// TIA Portal V19 export
FUNCTION "MODE SELECTION" : Void   // FC3, LAD
{ S7_Optimized_Access := 'TRUE' }
// stored: SetENOAutomatically false
   VAR_TEMP   // added for the SCL form of the ladder/FBD networks
      _w1 : Bool;
   END_VAR
BEGIN

REGION Network 1: STANDBY \///////////////////////////////// RO-1 ///////////////////////////////////////////
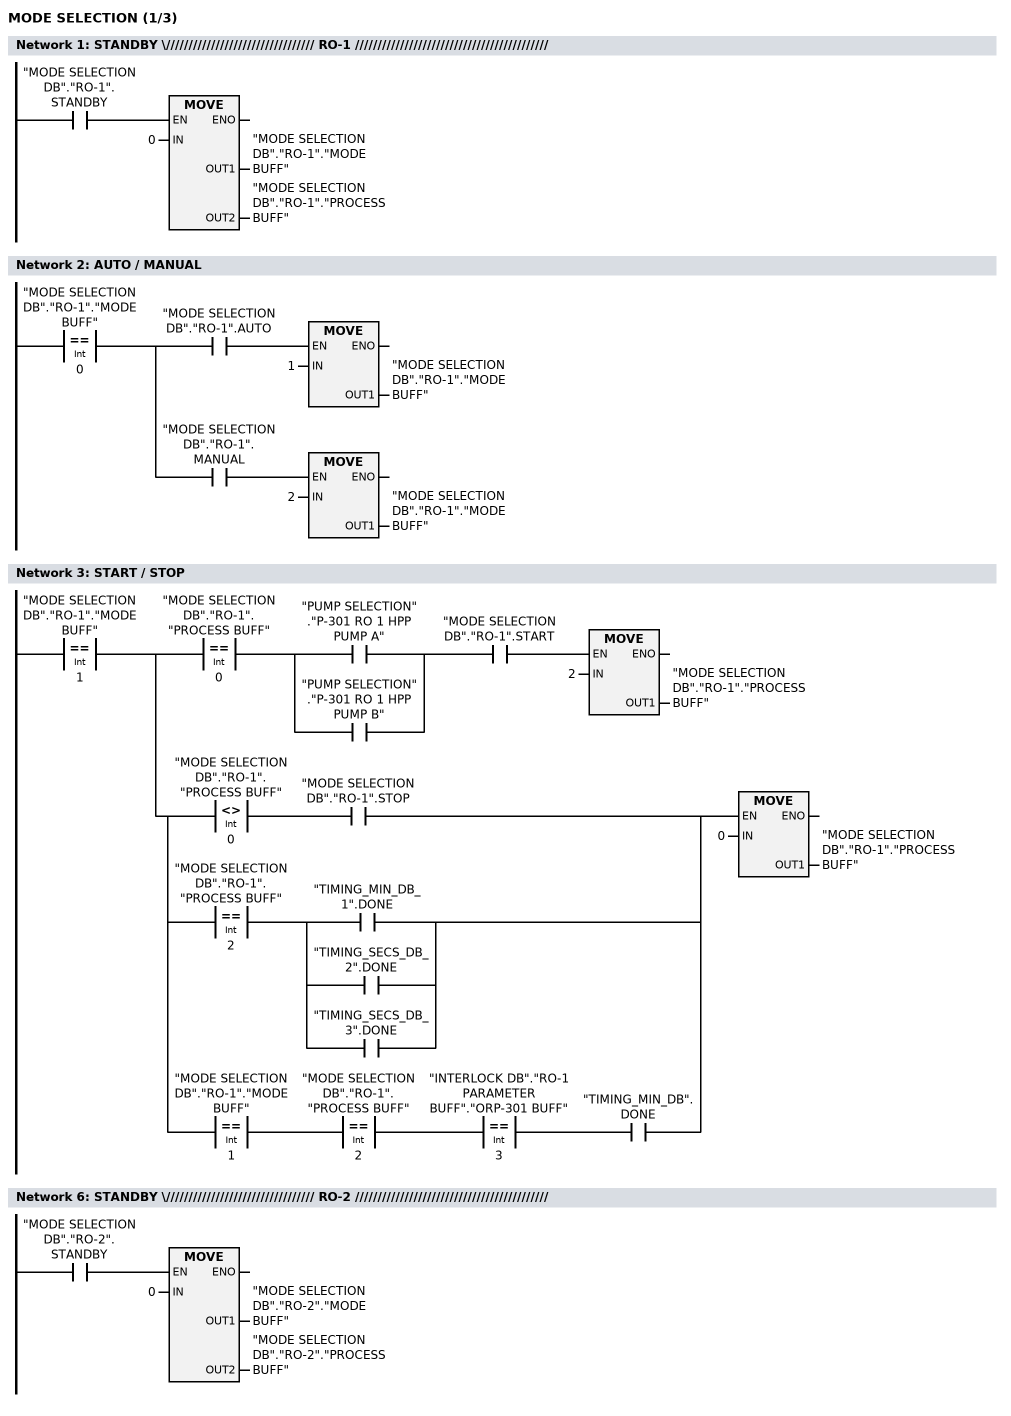
   RUNG wire#powerrail
      Contact( "MODE SELECTION DB"."RO-1".STANDBY )
      Move(in := 0, out1 => "MODE SELECTION DB"."RO-1"."MODE BUFF", out2 => "MODE SELECTION DB"."RO-1"."PROCESS BUFF")
   END_RUNG
   // the same network as SCL:
   IF "MODE SELECTION DB"."RO-1".STANDBY THEN
       "MODE SELECTION DB"."RO-1"."MODE BUFF" := 0;
       "MODE SELECTION DB"."RO-1"."PROCESS BUFF" := 0;
   END_IF;
END_REGION

REGION Network 2: AUTO / MANUAL
   RUNG wire#powerrail
      { S7_Templates := "SrcType := Int" } EQ_Contact(in1 := "MODE SELECTION DB"."RO-1"."MODE BUFF", in2 := 0)
      wire#w1
      Contact( "MODE SELECTION DB"."RO-1".AUTO )
      Move(in := 1, out1 => "MODE SELECTION DB"."RO-1"."MODE BUFF")
   END_RUNG
   RUNG wire#w1
      Contact( "MODE SELECTION DB"."RO-1".MANUAL )
      Move(in := 2, out1 => "MODE SELECTION DB"."RO-1"."MODE BUFF")
   END_RUNG
   // the same network as SCL:
   #_w1 := "MODE SELECTION DB"."RO-1"."MODE BUFF" = 0;
   IF #_w1 AND "MODE SELECTION DB"."RO-1".AUTO THEN "MODE SELECTION DB"."RO-1"."MODE BUFF" := 1; END_IF;
   IF #_w1 AND "MODE SELECTION DB"."RO-1".MANUAL THEN "MODE SELECTION DB"."RO-1"."MODE BUFF" := 2; END_IF;
END_REGION

REGION Network 3: START / STOP
   RUNG wire#powerrail
      { S7_Templates := "SrcType := Int" } EQ_Contact(in1 := "MODE SELECTION DB"."RO-1"."MODE BUFF", in2 := 1)
      wire#w1
      { S7_Templates := "SrcType := Int" } EQ_Contact(in1 := "MODE SELECTION DB"."RO-1"."PROCESS BUFF", in2 := 0)
      wire#w2
      Contact( "PUMP SELECTION"."P-301 RO 1 HPP PUMP A" )
      wire#w3
      Contact( "MODE SELECTION DB"."RO-1".START )
      Move(in := 2, out1 => "MODE SELECTION DB"."RO-1"."PROCESS BUFF")
   END_RUNG
   RUNG wire#w2
      Contact( "PUMP SELECTION"."P-301 RO 1 HPP PUMP B" )
   END_RUNG wire#w3
   RUNG wire#w1
      { S7_Templates := "SrcType := Int" } NE_Contact(in1 := "MODE SELECTION DB"."RO-1"."PROCESS BUFF", in2 := 0)
      Contact( "MODE SELECTION DB"."RO-1".STOP )
      wire#w4
      Move(in := 0, out1 => "MODE SELECTION DB"."RO-1"."PROCESS BUFF")
   END_RUNG
   RUNG wire#w1
      { S7_Templates := "SrcType := Int" } EQ_Contact(in1 := "MODE SELECTION DB"."RO-1"."PROCESS BUFF", in2 := 2)
      wire#w5
      Contact( "TIMING_MIN_DB_1".DONE )
   END_RUNG wire#w4
   RUNG wire#w5
      Contact( "TIMING_SECS_DB_2".DONE )
   END_RUNG wire#w4
   RUNG wire#w5
      Contact( "TIMING_SECS_DB_3".DONE )
   END_RUNG wire#w4
   RUNG wire#w1
      { S7_Templates := "SrcType := Int" } EQ_Contact(in1 := "MODE SELECTION DB"."RO-1"."MODE BUFF", in2 := 1)
      { S7_Templates := "SrcType := Int" } EQ_Contact(in1 := "MODE SELECTION DB"."RO-1"."PROCESS BUFF", in2 := 2)
      { S7_Templates := "SrcType := Int" } EQ_Contact(in1 := "INTERLOCK DB"."RO-1 PARAMETER BUFF"."ORP-301 BUFF", in2 := 3)
      Contact( "TIMING_MIN_DB".DONE )
   END_RUNG wire#w4
   // the same network as SCL:
   #_w1 := "MODE SELECTION DB"."RO-1"."MODE BUFF" = 1;
   IF #_w1 AND ("MODE SELECTION DB"."RO-1"."PROCESS BUFF" = 0) AND ("PUMP SELECTION"."P-301 RO 1 HPP PUMP A" OR "PUMP SELECTION"."P-301 RO 1 HPP PUMP B") AND "MODE SELECTION DB"."RO-1".START THEN
       "MODE SELECTION DB"."RO-1"."PROCESS BUFF" := 2;
   END_IF;
   IF #_w1 AND ((("MODE SELECTION DB"."RO-1"."PROCESS BUFF" <> 0) AND "MODE SELECTION DB"."RO-1".STOP) OR (("MODE SELECTION DB"."RO-1"."PROCESS BUFF" = 2) AND ("TIMING_MIN_DB_1".DONE OR "TIMING_SECS_DB_2".DONE OR "TIMING_SECS_DB_3".DONE)) OR (("MODE SELECTION DB"."RO-1"."MODE BUFF" = 1) AND ("MODE SELECTION DB"."RO-1"."PROCESS BUFF" = 2) AND ("INTERLOCK DB"."RO-1 PARAMETER BUFF"."ORP-301 BUFF" = 3) AND "TIMING_MIN_DB".DONE)) THEN
       "MODE SELECTION DB"."RO-1"."PROCESS BUFF" := 0;
   END_IF;
END_REGION

REGION Network 6: STANDBY \///////////////////////////////// RO-2 ///////////////////////////////////////////
   RUNG wire#powerrail
      Contact( "MODE SELECTION DB"."RO-2".STANDBY )
      Move(in := 0, out1 => "MODE SELECTION DB"."RO-2"."MODE BUFF", out2 => "MODE SELECTION DB"."RO-2"."PROCESS BUFF")
   END_RUNG
   // the same network as SCL:
   IF "MODE SELECTION DB"."RO-2".STANDBY THEN
       "MODE SELECTION DB"."RO-2"."MODE BUFF" := 0;
       "MODE SELECTION DB"."RO-2"."PROCESS BUFF" := 0;
   END_IF;
END_REGION

REGION Network 7: AUTO / MANUAL
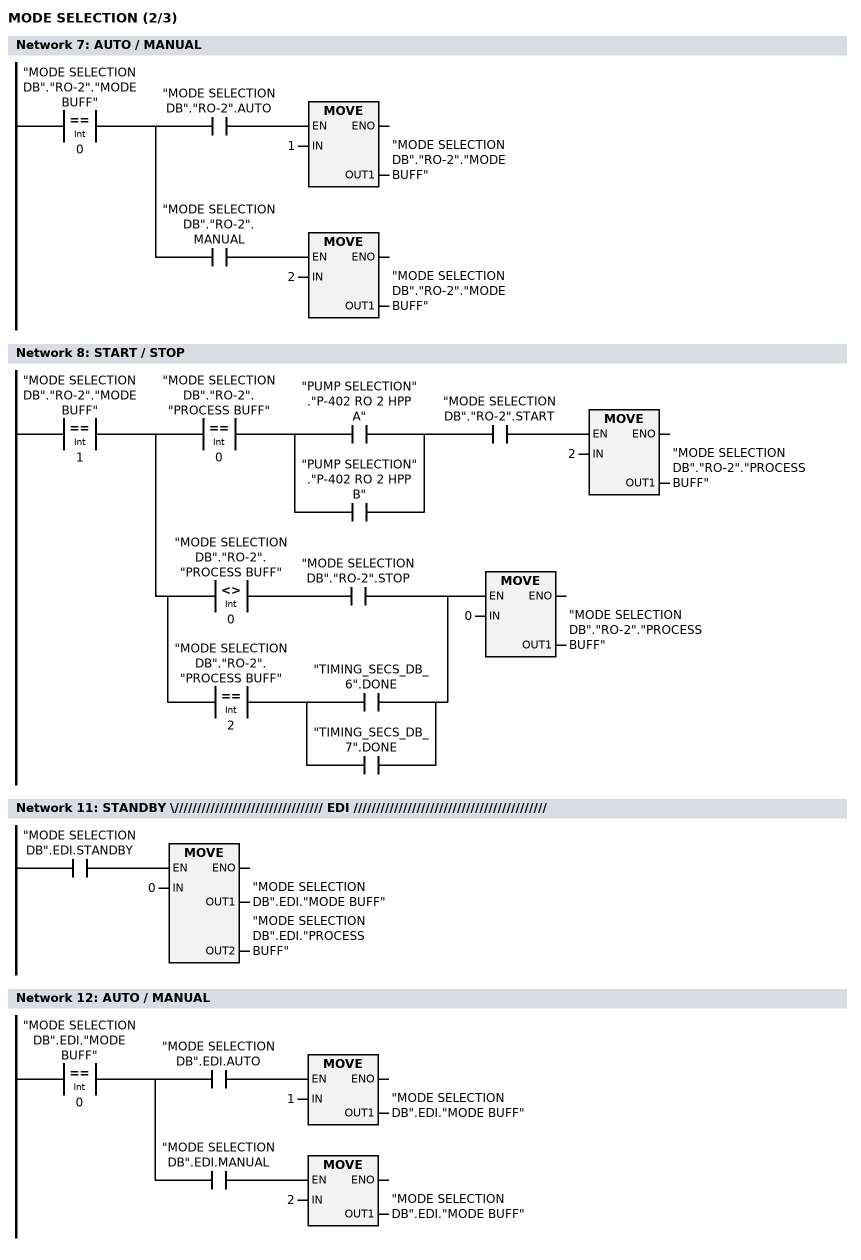
   RUNG wire#powerrail
      { S7_Templates := "SrcType := Int" } EQ_Contact(in1 := "MODE SELECTION DB"."RO-2"."MODE BUFF", in2 := 0)
      wire#w1
      Contact( "MODE SELECTION DB"."RO-2".AUTO )
      Move(in := 1, out1 => "MODE SELECTION DB"."RO-2"."MODE BUFF")
   END_RUNG
   RUNG wire#w1
      Contact( "MODE SELECTION DB"."RO-2".MANUAL )
      Move(in := 2, out1 => "MODE SELECTION DB"."RO-2"."MODE BUFF")
   END_RUNG
   // the same network as SCL:
   #_w1 := "MODE SELECTION DB"."RO-2"."MODE BUFF" = 0;
   IF #_w1 AND "MODE SELECTION DB"."RO-2".AUTO THEN "MODE SELECTION DB"."RO-2"."MODE BUFF" := 1; END_IF;
   IF #_w1 AND "MODE SELECTION DB"."RO-2".MANUAL THEN "MODE SELECTION DB"."RO-2"."MODE BUFF" := 2; END_IF;
END_REGION

REGION Network 8: START / STOP
   RUNG wire#powerrail
      { S7_Templates := "SrcType := Int" } EQ_Contact(in1 := "MODE SELECTION DB"."RO-2"."MODE BUFF", in2 := 1)
      wire#w1
      { S7_Templates := "SrcType := Int" } EQ_Contact(in1 := "MODE SELECTION DB"."RO-2"."PROCESS BUFF", in2 := 0)
      wire#w2
      Contact( "PUMP SELECTION"."P-402 RO 2 HPP A" )
      wire#w3
      Contact( "MODE SELECTION DB"."RO-2".START )
      Move(in := 2, out1 => "MODE SELECTION DB"."RO-2"."PROCESS BUFF")
   END_RUNG
   RUNG wire#w2
      Contact( "PUMP SELECTION"."P-402 RO 2 HPP B" )
   END_RUNG wire#w3
   RUNG wire#w1
      { S7_Templates := "SrcType := Int" } NE_Contact(in1 := "MODE SELECTION DB"."RO-2"."PROCESS BUFF", in2 := 0)
      Contact( "MODE SELECTION DB"."RO-2".STOP )
      wire#w4
      Move(in := 0, out1 => "MODE SELECTION DB"."RO-2"."PROCESS BUFF")
   END_RUNG
   RUNG wire#w1
      { S7_Templates := "SrcType := Int" } EQ_Contact(in1 := "MODE SELECTION DB"."RO-2"."PROCESS BUFF", in2 := 2)
      wire#w5
      Contact( "TIMING_SECS_DB_6".DONE )
   END_RUNG wire#w4
   RUNG wire#w5
      Contact( "TIMING_SECS_DB_7".DONE )
   END_RUNG wire#w4
   // the same network as SCL:
   #_w1 := "MODE SELECTION DB"."RO-2"."MODE BUFF" = 1;
   IF #_w1 AND ("MODE SELECTION DB"."RO-2"."PROCESS BUFF" = 0) AND ("PUMP SELECTION"."P-402 RO 2 HPP A" OR "PUMP SELECTION"."P-402 RO 2 HPP B") AND "MODE SELECTION DB"."RO-2".START THEN
       "MODE SELECTION DB"."RO-2"."PROCESS BUFF" := 2;
   END_IF;
   IF #_w1 AND ((("MODE SELECTION DB"."RO-2"."PROCESS BUFF" <> 0) AND "MODE SELECTION DB"."RO-2".STOP) OR (("MODE SELECTION DB"."RO-2"."PROCESS BUFF" = 2) AND ("TIMING_SECS_DB_6".DONE OR "TIMING_SECS_DB_7".DONE))) THEN
       "MODE SELECTION DB"."RO-2"."PROCESS BUFF" := 0;
   END_IF;
END_REGION

REGION Network 11: STANDBY \///////////////////////////////// EDI ///////////////////////////////////////////
   RUNG wire#powerrail
      Contact( "MODE SELECTION DB".EDI.STANDBY )
      Move(in := 0, out1 => "MODE SELECTION DB".EDI."MODE BUFF", out2 => "MODE SELECTION DB".EDI."PROCESS BUFF")
   END_RUNG
   // the same network as SCL:
   IF "MODE SELECTION DB".EDI.STANDBY THEN
       "MODE SELECTION DB".EDI."MODE BUFF" := 0;
       "MODE SELECTION DB".EDI."PROCESS BUFF" := 0;
   END_IF;
END_REGION

REGION Network 12: AUTO / MANUAL
   RUNG wire#powerrail
      { S7_Templates := "SrcType := Int" } EQ_Contact(in1 := "MODE SELECTION DB".EDI."MODE BUFF", in2 := 0)
      wire#w1
      Contact( "MODE SELECTION DB".EDI.AUTO )
      Move(in := 1, out1 => "MODE SELECTION DB".EDI."MODE BUFF")
   END_RUNG
   RUNG wire#w1
      Contact( "MODE SELECTION DB".EDI.MANUAL )
      Move(in := 2, out1 => "MODE SELECTION DB".EDI."MODE BUFF")
   END_RUNG
   // the same network as SCL:
   #_w1 := "MODE SELECTION DB".EDI."MODE BUFF" = 0;
   IF #_w1 AND "MODE SELECTION DB".EDI.AUTO THEN "MODE SELECTION DB".EDI."MODE BUFF" := 1; END_IF;
   IF #_w1 AND "MODE SELECTION DB".EDI.MANUAL THEN "MODE SELECTION DB".EDI."MODE BUFF" := 2; END_IF;
END_REGION

REGION Network 13: START / STOP
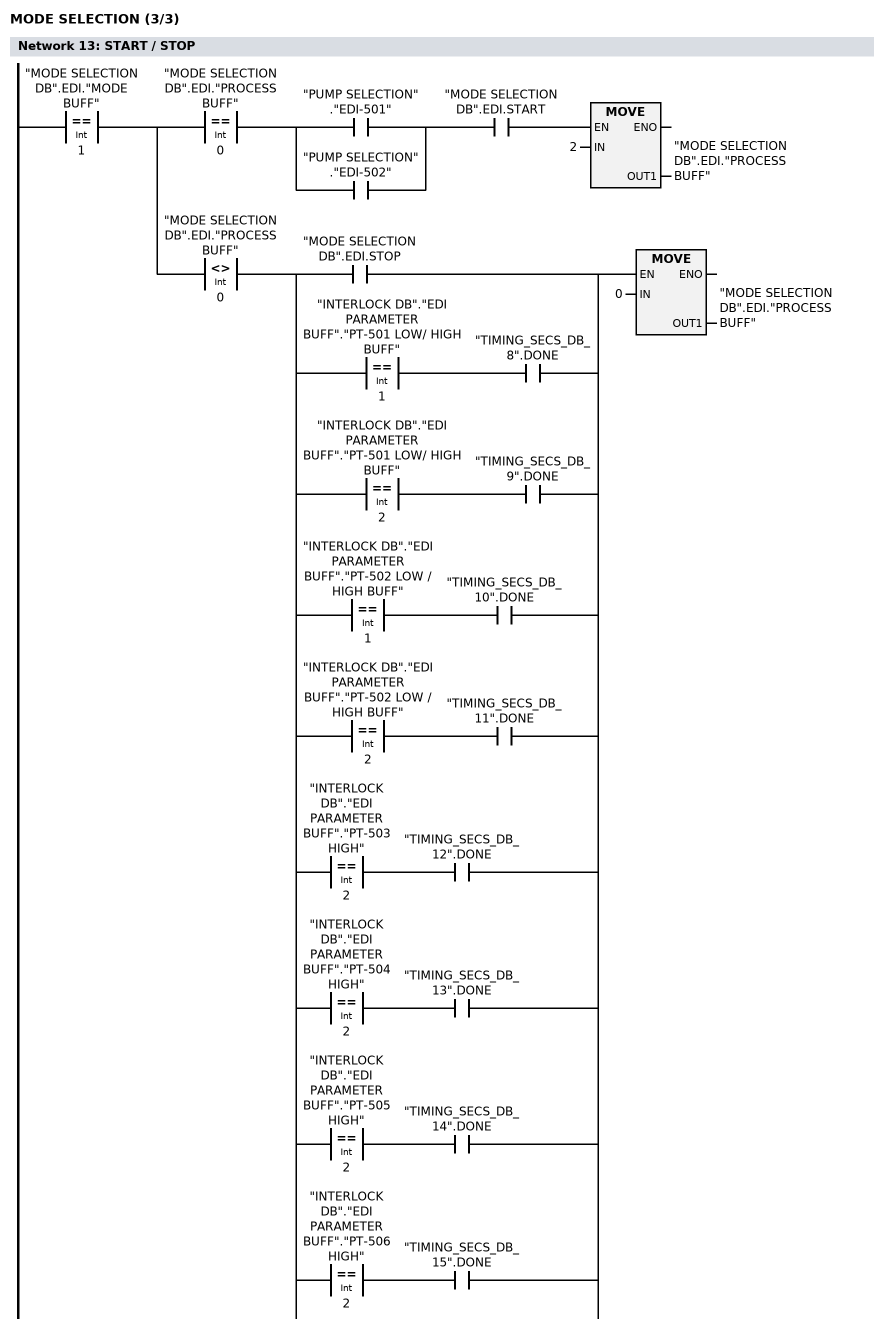
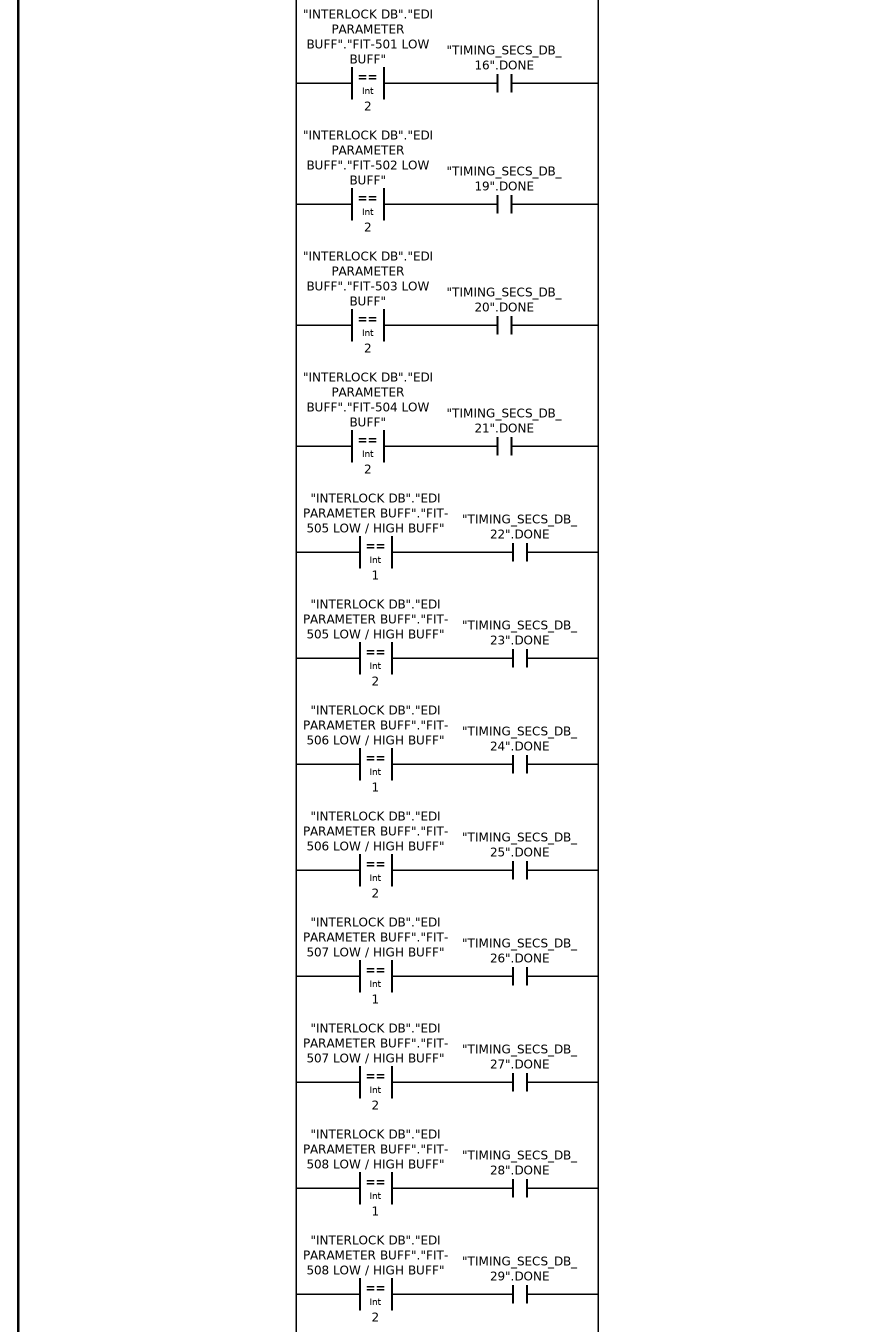
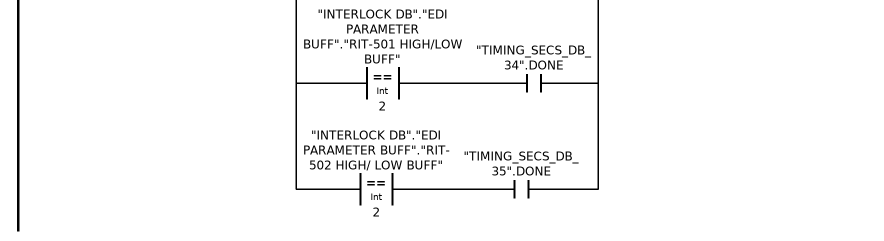
   RUNG wire#powerrail
      { S7_Templates := "SrcType := Int" } EQ_Contact(in1 := "MODE SELECTION DB".EDI."MODE BUFF", in2 := 1)
      wire#w1
      { S7_Templates := "SrcType := Int" } EQ_Contact(in1 := "MODE SELECTION DB".EDI."PROCESS BUFF", in2 := 0)
      wire#w2
      Contact( "PUMP SELECTION"."EDI-501" )
      wire#w3
      Contact( "MODE SELECTION DB".EDI.START )
      Move(in := 2, out1 => "MODE SELECTION DB".EDI."PROCESS BUFF")
   END_RUNG
   RUNG wire#w2
      Contact( "PUMP SELECTION"."EDI-502" )
   END_RUNG wire#w3
   RUNG wire#w1
      { S7_Templates := "SrcType := Int" } NE_Contact(in1 := "MODE SELECTION DB".EDI."PROCESS BUFF", in2 := 0)
      wire#w4
      Contact( "MODE SELECTION DB".EDI.STOP )
      wire#w5
      Move(in := 0, out1 => "MODE SELECTION DB".EDI."PROCESS BUFF")
   END_RUNG
   RUNG wire#w4
      { S7_Templates := "SrcType := Int" } EQ_Contact(in1 := "INTERLOCK DB"."EDI PARAMETER BUFF"."PT-501 LOW/ HIGH BUFF", in2 := 1)
      Contact( "TIMING_SECS_DB_8".DONE )
   END_RUNG wire#w5
   RUNG wire#w4
      { S7_Templates := "SrcType := Int" } EQ_Contact(in1 := "INTERLOCK DB"."EDI PARAMETER BUFF"."PT-501 LOW/ HIGH BUFF", in2 := 2)
      Contact( "TIMING_SECS_DB_9".DONE )
   END_RUNG wire#w5
   RUNG wire#w4
      { S7_Templates := "SrcType := Int" } EQ_Contact(in1 := "INTERLOCK DB"."EDI PARAMETER BUFF"."PT-502 LOW / HIGH BUFF", in2 := 1)
      Contact( "TIMING_SECS_DB_10".DONE )
   END_RUNG wire#w5
   RUNG wire#w4
      { S7_Templates := "SrcType := Int" } EQ_Contact(in1 := "INTERLOCK DB"."EDI PARAMETER BUFF"."PT-502 LOW / HIGH BUFF", in2 := 2)
      Contact( "TIMING_SECS_DB_11".DONE )
   END_RUNG wire#w5
   RUNG wire#w4
      { S7_Templates := "SrcType := Int" } EQ_Contact(in1 := "INTERLOCK DB"."EDI PARAMETER BUFF"."PT-503 HIGH", in2 := 2)
      Contact( "TIMING_SECS_DB_12".DONE )
   END_RUNG wire#w5
   RUNG wire#w4
      { S7_Templates := "SrcType := Int" } EQ_Contact(in1 := "INTERLOCK DB"."EDI PARAMETER BUFF"."PT-504 HIGH", in2 := 2)
      Contact( "TIMING_SECS_DB_13".DONE )
   END_RUNG wire#w5
   RUNG wire#w4
      { S7_Templates := "SrcType := Int" } EQ_Contact(in1 := "INTERLOCK DB"."EDI PARAMETER BUFF"."PT-505 HIGH", in2 := 2)
      Contact( "TIMING_SECS_DB_14".DONE )
   END_RUNG wire#w5
   RUNG wire#w4
      { S7_Templates := "SrcType := Int" } EQ_Contact(in1 := "INTERLOCK DB"."EDI PARAMETER BUFF"."PT-506 HIGH", in2 := 2)
      Contact( "TIMING_SECS_DB_15".DONE )
   END_RUNG wire#w5
   RUNG wire#w4
      { S7_Templates := "SrcType := Int" } EQ_Contact(in1 := "INTERLOCK DB"."EDI PARAMETER BUFF"."FIT-501 LOW BUFF", in2 := 2)
      Contact( "TIMING_SECS_DB_16".DONE )
   END_RUNG wire#w5
   RUNG wire#w4
      { S7_Templates := "SrcType := Int" } EQ_Contact(in1 := "INTERLOCK DB"."EDI PARAMETER BUFF"."FIT-502 LOW  BUFF", in2 := 2)
      Contact( "TIMING_SECS_DB_19".DONE )
   END_RUNG wire#w5
   RUNG wire#w4
      { S7_Templates := "SrcType := Int" } EQ_Contact(in1 := "INTERLOCK DB"."EDI PARAMETER BUFF"."FIT-503 LOW BUFF", in2 := 2)
      Contact( "TIMING_SECS_DB_20".DONE )
   END_RUNG wire#w5
   RUNG wire#w4
      { S7_Templates := "SrcType := Int" } EQ_Contact(in1 := "INTERLOCK DB"."EDI PARAMETER BUFF"."FIT-504 LOW BUFF", in2 := 2)
      Contact( "TIMING_SECS_DB_21".DONE )
   END_RUNG wire#w5
   RUNG wire#w4
      { S7_Templates := "SrcType := Int" } EQ_Contact(in1 := "INTERLOCK DB"."EDI PARAMETER BUFF"."FIT-505 LOW / HIGH BUFF", in2 := 1)
      Contact( "TIMING_SECS_DB_22".DONE )
   END_RUNG wire#w5
   RUNG wire#w4
      { S7_Templates := "SrcType := Int" } EQ_Contact(in1 := "INTERLOCK DB"."EDI PARAMETER BUFF"."FIT-505 LOW / HIGH BUFF", in2 := 2)
      Contact( "TIMING_SECS_DB_23".DONE )
   END_RUNG wire#w5
   RUNG wire#w4
      { S7_Templates := "SrcType := Int" } EQ_Contact(in1 := "INTERLOCK DB"."EDI PARAMETER BUFF"."FIT-506 LOW / HIGH BUFF", in2 := 1)
      Contact( "TIMING_SECS_DB_24".DONE )
   END_RUNG wire#w5
   RUNG wire#w4
      { S7_Templates := "SrcType := Int" } EQ_Contact(in1 := "INTERLOCK DB"."EDI PARAMETER BUFF"."FIT-506 LOW / HIGH BUFF", in2 := 2)
      Contact( "TIMING_SECS_DB_25".DONE )
   END_RUNG wire#w5
   RUNG wire#w4
      { S7_Templates := "SrcType := Int" } EQ_Contact(in1 := "INTERLOCK DB"."EDI PARAMETER BUFF"."FIT-507 LOW / HIGH BUFF", in2 := 1)
      Contact( "TIMING_SECS_DB_26".DONE )
   END_RUNG wire#w5
   RUNG wire#w4
      { S7_Templates := "SrcType := Int" } EQ_Contact(in1 := "INTERLOCK DB"."EDI PARAMETER BUFF"."FIT-507 LOW / HIGH BUFF", in2 := 2)
      Contact( "TIMING_SECS_DB_27".DONE )
   END_RUNG wire#w5
   RUNG wire#w4
      { S7_Templates := "SrcType := Int" } EQ_Contact(in1 := "INTERLOCK DB"."EDI PARAMETER BUFF"."FIT-508 LOW / HIGH BUFF", in2 := 1)
      Contact( "TIMING_SECS_DB_28".DONE )
   END_RUNG wire#w5
   RUNG wire#w4
      { S7_Templates := "SrcType := Int" } EQ_Contact(in1 := "INTERLOCK DB"."EDI PARAMETER BUFF"."FIT-508 LOW / HIGH BUFF", in2 := 2)
      Contact( "TIMING_SECS_DB_29".DONE )
   END_RUNG wire#w5
   RUNG wire#w4
      { S7_Templates := "SrcType := Int" } EQ_Contact(in1 := "INTERLOCK DB"."EDI PARAMETER BUFF"."RIT-501 HIGH/LOW BUFF", in2 := 2)
      Contact( "TIMING_SECS_DB_34".DONE )
   END_RUNG wire#w5
   RUNG wire#w4
      { S7_Templates := "SrcType := Int" } EQ_Contact(in1 := "INTERLOCK DB"."EDI PARAMETER BUFF"."RIT-502 HIGH/ LOW BUFF", in2 := 2)
      Contact( "TIMING_SECS_DB_35".DONE )
   END_RUNG wire#w5
   // the same network as SCL:
   #_w1 := "MODE SELECTION DB".EDI."MODE BUFF" = 1;
   IF #_w1 AND ("MODE SELECTION DB".EDI."PROCESS BUFF" = 0) AND ("PUMP SELECTION"."EDI-501" OR "PUMP SELECTION"."EDI-502") AND "MODE SELECTION DB".EDI.START THEN
       "MODE SELECTION DB".EDI."PROCESS BUFF" := 2;
   END_IF;
   IF #_w1 AND ("MODE SELECTION DB".EDI."PROCESS BUFF" <> 0) AND ("MODE SELECTION DB".EDI.STOP OR (("INTERLOCK DB"."EDI PARAMETER BUFF"."PT-501 LOW/ HIGH BUFF" = 1) AND "TIMING_SECS_DB_8".DONE) OR (("INTERLOCK DB"."EDI PARAMETER BUFF"."PT-501 LOW/ HIGH BUFF" = 2) AND "TIMING_SECS_DB_9".DONE) OR (("INTERLOCK DB"."EDI PARAMETER BUFF"."PT-502 LOW / HIGH BUFF" = 1) AND "TIMING_SECS_DB_10".DONE) OR (("INTERLOCK DB"."EDI PARAMETER BUFF"."PT-502 LOW / HIGH BUFF" = 2) AND "TIMING_SECS_DB_11".DONE) OR (("INTERLOCK DB"."EDI PARAMETER BUFF"."PT-503 HIGH" = 2) AND "TIMING_SECS_DB_12".DONE) OR (("INTERLOCK DB"."EDI PARAMETER BUFF"."PT-504 HIGH" = 2) AND "TIMING_SECS_DB_13".DONE) OR (("INTERLOCK DB"."EDI PARAMETER BUFF"."PT-505 HIGH" = 2) AND "TIMING_SECS_DB_14".DONE) OR (("INTERLOCK DB"."EDI PARAMETER BUFF"."PT-506 HIGH" = 2) AND "TIMING_SECS_DB_15".DONE) OR (("INTERLOCK DB"."EDI PARAMETER BUFF"."FIT-501 LOW BUFF" = 2) AND "TIMING_SECS_DB_16".DONE) OR (("INTERLOCK DB"."EDI PARAMETER BUFF"."FIT-502 LOW  BUFF" = 2) AND "TIMING_SECS_DB_19".DONE) OR (("INTERLOCK DB"."EDI PARAMETER BUFF"."FIT-503 LOW BUFF" = 2) AND "TIMING_SECS_DB_20".DONE) OR (("INTERLOCK DB"."EDI PARAMETER BUFF"."FIT-504 LOW BUFF" = 2) AND "TIMING_SECS_DB_21".DONE) OR (("INTERLOCK DB"."EDI PARAMETER BUFF"."FIT-505 LOW / HIGH BUFF" = 1) AND "TIMING_SECS_DB_22".DONE) OR (("INTERLOCK DB"."EDI PARAMETER BUFF"."FIT-505 LOW / HIGH BUFF" = 2) AND "TIMING_SECS_DB_23".DONE) OR (("INTERLOCK DB"."EDI PARAMETER BUFF"."FIT-506 LOW / HIGH BUFF" = 1) AND "TIMING_SECS_DB_24".DONE) OR (("INTERLOCK DB"."EDI PARAMETER BUFF"."FIT-506 LOW / HIGH BUFF" = 2) AND "TIMING_SECS_DB_25".DONE) OR (("INTERLOCK DB"."EDI PARAMETER BUFF"."FIT-507 LOW / HIGH BUFF" = 1) AND "TIMING_SECS_DB_26".DONE) OR (("INTERLOCK DB"."EDI PARAMETER BUFF"."FIT-507 LOW / HIGH BUFF" = 2) AND "TIMING_SECS_DB_27".DONE) OR (("INTERLOCK DB"."EDI PARAMETER BUFF"."FIT-508 LOW / HIGH BUFF" = 1) AND "TIMING_SECS_DB_28".DONE) OR (("INTERLOCK DB"."EDI PARAMETER BUFF"."FIT-508 LOW / HIGH BUFF" = 2) AND "TIMING_SECS_DB_29".DONE) OR (("INTERLOCK DB"."EDI PARAMETER BUFF"."RIT-501 HIGH/LOW BUFF" = 2) AND "TIMING_SECS_DB_34".DONE) OR (("INTERLOCK DB"."EDI PARAMETER BUFF"."RIT-502 HIGH/ LOW BUFF" = 2) AND "TIMING_SECS_DB_35".DONE)) THEN
       "MODE SELECTION DB".EDI."PROCESS BUFF" := 0;
   END_IF;
END_REGION
END_FUNCTION
